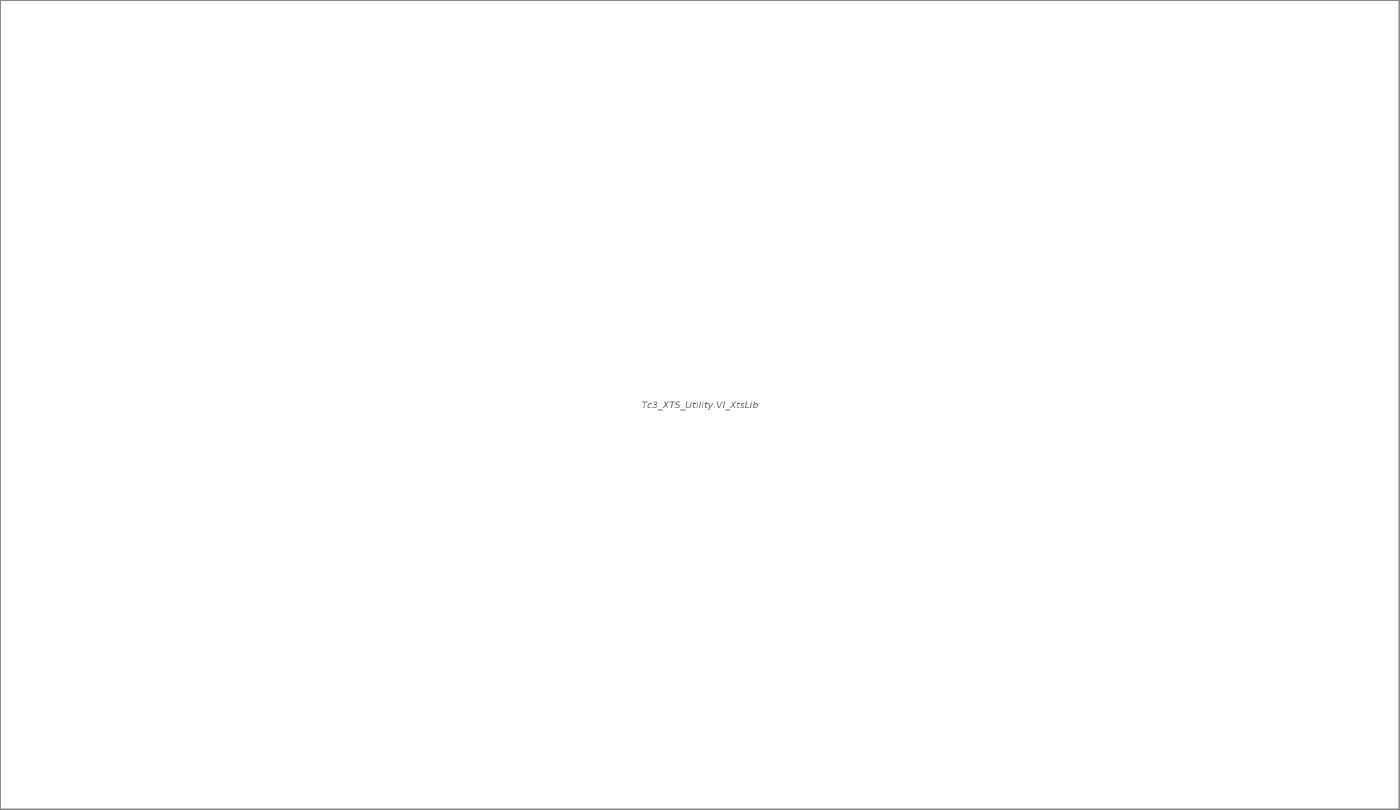
VISUALIZATION PageXtsDiagnostic_1  // 1520x880
    Frame (0,0 1520x880)
        shows Tc3_XTS_Utility.VI_XtsLib()
END_VISUALIZATION

(* stored: Version 1.1.0.1, ProductVersion 3.1.4024.12
   Visu PageXtsDiagnostic_1: Id {cf35a50f-fdfb-47dc-acb6-97f8017fb35d} *)
